GLOBALCONSTANTS PKP_2200 (* Global constants *)
  (* Standard: 61499-1 *)
  (* Version 1.0, 2023-10-22, franz *)
  VAR_GLOBAL CONSTANT
    PKP_2200_DEFAULT : USINT := USINT#16#21;
  END_VAR
END_GLOBALCONSTANTS
